// SIMATIC S7-200 SMART project (STEP 7-Micro/WIN SMART), CPU SR40

SYMBOL_TABLE 系统符号
Clock_1s         SM0.5    // 针对 1 s 的周期时间，时钟脉冲接通 0.5 s，断开 0.5 s.
END_SYMBOL_TABLE

ORGANIZATION_BLOCK MAIN:OB1
TITLE=程序注释
BEGIN
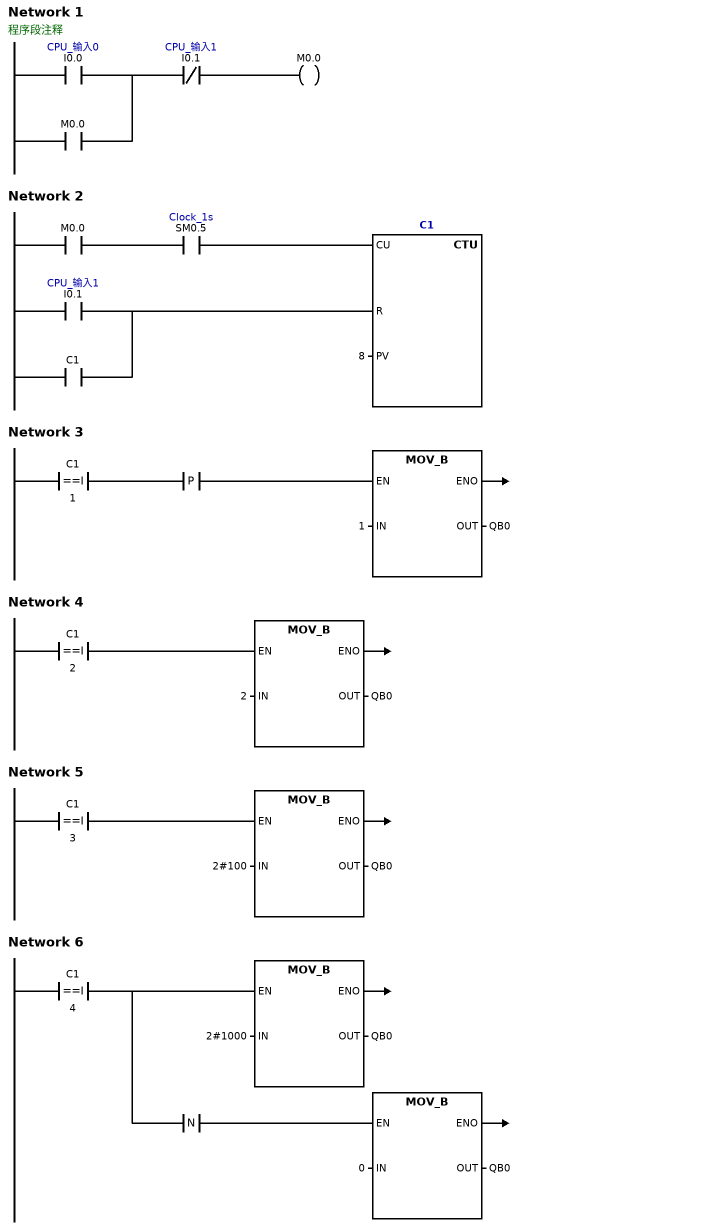
Network 1
// 程序段注释
LD     CPU_输入0:I0.0
O      M0.0
AN     CPU_输入1:I0.1
=      M0.0
Network 2
LD     M0.0
A      Clock_1s:SM0.5
LD     CPU_输入1:I0.1
O      C1
CTU    C1, 8
Network 3
LDW=   C1, 1
EU
MOVB   1, QB0
Network 4
LDW=   C1, 2
MOVB   2, QB0
Network 5
LDW=   C1, 3
MOVB   2#100, QB0
Network 6
LDW=   C1, 4
MOVB   2#1000, QB0
ED
MOVB   0, QB0
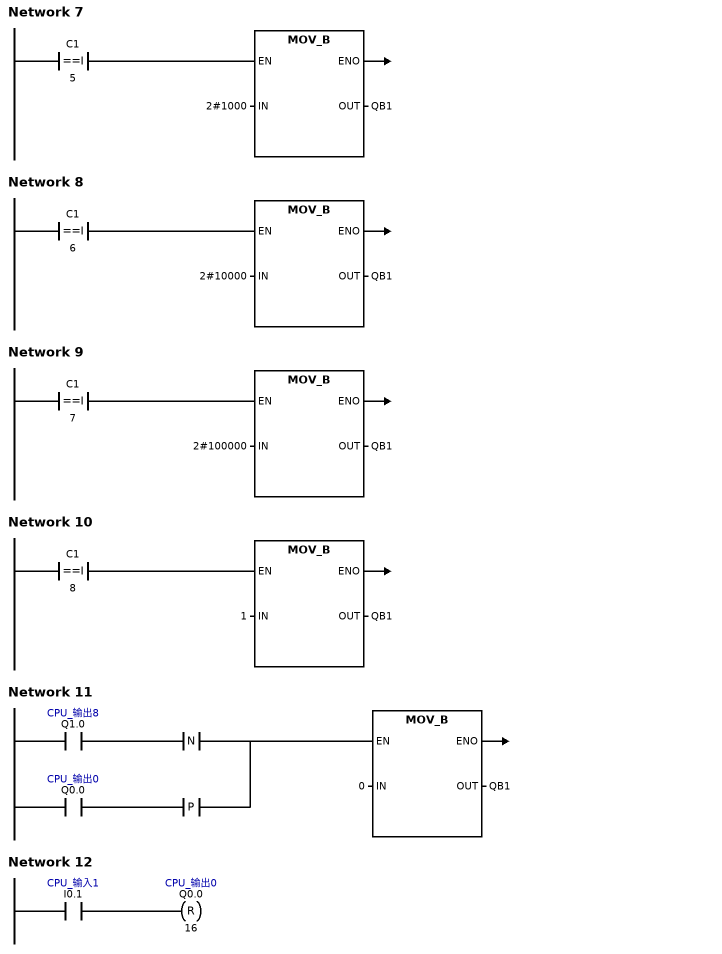
Network 7
LDW=   C1, 5
MOVB   2#1000, QB1
Network 8
LDW=   C1, 6
MOVB   2#10000, QB1
Network 9
LDW=   C1, 7
MOVB   2#100000, QB1
Network 10
LDW=   C1, 8
MOVB   1, QB1
Network 11
LD     CPU_输出8:Q1.0
ED
LD     CPU_输出0:Q0.0
EU
OLD
MOVB   0, QB1
Network 12
LD     CPU_输入1:I0.1
R      CPU_输出0:Q0.0, 16
END_ORGANIZATION_BLOCK
